(* PLC project M3_17, Desconocido M3_17 1 *)
(* stored: creationDateTime 2025-06-09T23:37:46, modificationDateTime 2025-06-09T23:47:57 *)

PROGRAM Main
  VAR
    CTU0 : CTU;
    R_TRIG0 : R_TRIG;
    xSensorCaja : BOOL;
    xActivarPaletizado : BOOL;
    xProcesoPaletizado : BOOL;
    xPaletizadoTerminado : BOOL;
  END_VAR
  VAR  (* added by the conversion: wires and edge detectors of the diagram *)
    R_TRIG1 : R_TRIG;
  END_VAR

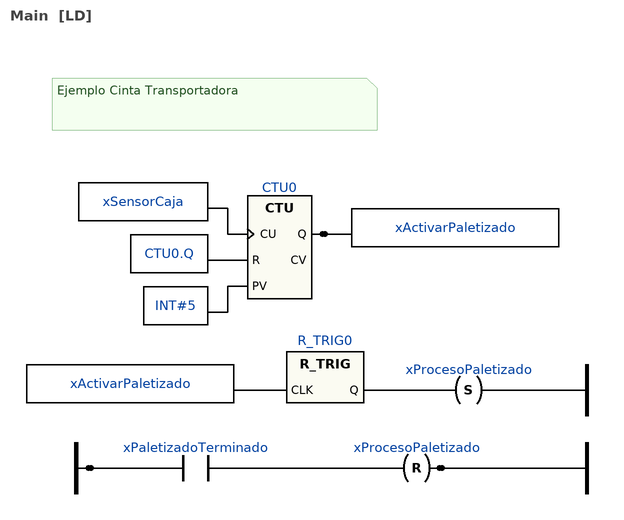
(* LD diagram, written out as Structured Text *)
(* Ejemplo Cinta Transportadora *)
R_TRIG1(CLK := xSensorCaja);
CTU0(CU := R_TRIG1.Q, R := CTU0.Q, PV := INT#5);
xActivarPaletizado := CTU0.Q;
R_TRIG0(CLK := xActivarPaletizado);
IF R_TRIG0.Q THEN xProcesoPaletizado := TRUE; END_IF;
IF xPaletizadoTerminado THEN xProcesoPaletizado := FALSE; END_IF;
END_PROGRAM

CONFIGURATION Config0
  RESOURCE Res0 ON PLC
    TASK task0(INTERVAL := T#20ms, PRIORITY := 0);
    PROGRAM instance0 WITH task0 : Main;
  END_RESOURCE
END_CONFIGURATION
